ABB RobotStudio station: CameraLegos_20180405-085602.rsstn

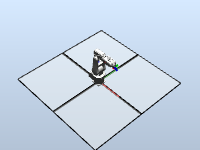
Station CameraLegos (saved by RobotStudio 6.6.7701.1025)
Controller System1
  mechanical unit ROB_1: IRB120_3_58__01, 6 joints, base frame (0, 0, 0) mm
Layout (positions relative to the parent item):
  - IRB120_3_58__01 [mechanism, from Robots\IRB120_3_58_G_01.rslib] at (0, 0, 0) mm; joint values [0, 0, 0, 0, 0.5236, 0] (rad or m)
  - MoveToViewpoint [smart component, from Components\MoveToViewpoint.rslib]
      properties: Viewpoint=(none); Time=0
  - Camera [smart component, from Components\Camera.rslib]
      properties: Path=; File Name=
Station logic (signal -> signal, property => property):
  MoveToViewpoint.Executed -> Camera.Execute
Targets, tools, work objects and paths stored in the station, written as RAPID:
! task T_ROB1
MODULE FunctionHandler
  PERS tooldata defaultTool:=[TRUE,[[0,0,0],[1,0,0,0]],[1,[0,0,0.001],[1,0,0,0],0,0,0]];
  PERS wobjdata defaultWobj:=[FALSE,TRUE,"",[[0,0,0],[1,0,0,0]],[[0,0,0],[1,0,0,0]]];
  VAR signaldo defaultTakePictureActivationIO;
  VAR signaldi defaultTakePictureExecutedIO;
  PROC FH_TakePicture()
    SetDO defaultTakePictureActivationIO,1;
    WaitDI defaultTakePictureExecutedIO,1;
    SetDO defaultTakePictureActivationIO,0;
  ENDPROC
ENDMODULE

! task T_ROB1
MODULE CommandHandler
  PROC COMH_CommandListener()
  ENDPROC
ENDMODULE

! task T_ROB1
MODULE MatlabCamera
  PROC main()
    IP_Initialize;
    COMH_CommandListener;
  ENDPROC
ENDMODULE

! task T_ROB1
MODULE InitParameters
  PROC IP_Initialize()
    ConfL \Off;
    ConfJ \Off;
  ENDPROC
ENDMODULE

